FUNCTION_BLOCK FB_Logger EXTENDS FB_TcLogger
VAR
END_VAR

// Log events to the Visual Studio

METHOD M_Log
VAR_INPUT
	stEvent	: 		ST_Event;
END_VAR

VAR
	sMessage:			STRING(255);
END_VAR
IF stEvent.Active THEN
	sMessage:= Concat(Concat(stEvent.Instance, ' | iLogger = 0 | '), stEvent.Message);
	CASE stEvent.EventType OF
		E_Event.Error:
			ADSLOGSTR( msgCtrlMask := ADSLOG_MSGTYPE_ERROR , msgFmtStr := '%s', strArg := sMessage);
		E_Event.Warning:
			ADSLOGSTR( msgCtrlMask := ADSLOG_MSGTYPE_WARN , msgFmtStr := '%s', strArg := sMessage);
		E_Event.Information:
			ADSLOGSTR( msgCtrlMask := ADSLOG_MSGTYPE_HINT , msgFmtStr := '%s', strArg := sMessage);
		E_Event.Debug:
			ADSLOGSTR( msgCtrlMask := ADSLOG_MSGTYPE_HINT, msgFmtStr := '%s', strArg := sMessage);
		E_Event.Verbose:
			ADSLOGSTR( msgCtrlMask := ADSLOG_MSGTYPE_HINT , msgFmtStr := '%s', strArg := sMessage);
	END_CASE	
END_IF
END_METHOD

END_FUNCTION_BLOCK

(* stored: Version 1.1.0.1
   POU FB_Logger: Id {e1e358e0-2104-0577-0348-94cd81bffe81}, SpecialFunc None
   Method M_Log: Id {9e2c1dc1-68d4-0b75-365d-62c1554c8296} *)
